/// container for all communication data types that are used by the unit
TYPE AssemblyComRef :
STRUCT
  Publish : REFERENCE TO AssemblyComPublish; 
  Subscribe : REFERENCE TO AssemblyComSubscribe; 
END_STRUCT
END_TYPE

(* stored: Version 1.1.0.1
   DUT AssemblyComRef: Id {98f16b6f-19d9-4509-9cce-a841e41ee437} *)
